// Mitsubishi GX Works2 project: auotomatation project   PLC: FX3G

// global labels: Global1
VAR_GLOBAL
  start_day AT X007 : BOOL;
  stock_oats AT D1100 : REAL;
  oats_input AT D1105 : REAL;
  stock_protein AT D2100 : REAL;
  protein_input AT D2105 : REAL;
  stock_honey AT D3100 : REAL;
  honey_input AT D3105 : REAL;
END_VAR
VAR_GLOBAL CONSTANT
  oats_min_need : REAL := 400;
  protein_min_need : REAL := 320;
  honey_min_need : REAL := 160;
END_VAR
VAR_GLOBAL
  enough_stock AT M1 : BOOL;
  valid_input AT M5 : BOOL;
  working AT Y000 : BOOL;
  emergency AT X005 : BOOL;
  Sample AT X003 : BOOL;
  Bar_Type AT D1160 : REAL;
END_VAR
VAR_GLOBAL CONSTANT
  Protein_Max : REAL := 10.0;
  Protein_Min : REAL := 5.0;
  Basic_Max : REAL := 5.0;
  Basic_Min : REAL;
END_VAR
VAR_GLOBAL
  Protein_Is_More_Beautiful AT M3 : BOOL;
  Basic_Is_Beautiful AT M4 : BOOL;
  MixingTime AT TC1 : BOOL;
END_VAR
VAR_GLOBAL CONSTANT
  MixingDuration : INT := 50;
END_VAR
VAR_GLOBAL
  EndMixing AT TS1 : BOOL;
  KeepOnMixingBaby AT Y003 : BOOL;
END_VAR
VAR_GLOBAL CONSTANT
  OATFOR8 : REAL := 400;
  OATFOR8PROTEIN : REAL := 240.0;
  ProteinFor8BASIC : REAL := 160.0;
  ProteinFor8 : REAL := 320.0;
  HoneyFor8Basic : REAL := 120.0;
  HoneyFor8 : REAL := 160.0;
  MixingFor8Basic : REAL := 680.0;
  MixingFor8Protein : REAL := 720.0;
END_VAR
VAR_GLOBAL
  MixingContainer AT D1150 : REAL;
  StartBake AT X002 : BOOL;
  BakeContainer AT D1170 : REAL;
  TimeForBakingB AT TC2 : BOOL;
  TimeForBakingP AT TC3 : BOOL;
  FinishBakingBasic AT TS2 : BOOL;
  FinishBakingProtein AT TS3 : BOOL;
  BlinkAssist AT M11 : BOOL;
  FirstLight AT TS4 : BOOL;
  Sirugin1 AT TC4 : BOOL;
  FirstBake AT Y001 : BOOL;
END_VAR
VAR_GLOBAL CONSTANT
  Sirugin : INT := 6;
END_VAR
VAR_GLOBAL
  Sirugin2 AT TC5 : BOOL;
  SecondLight AT TS5 : BOOL;
  SecondBake AT Y002 : BOOL;
  StartPacking AT X006 : BOOL;
  PackOneBar AT X000 : BOOL;
  CountFirstBar AT CC0 : BOOL;
END_VAR
VAR_GLOBAL CONSTANT
  CountedFirstBar : INT := 1;
END_VAR
VAR_GLOBAL
  Count8Bars AT CC1 : BOOL;
END_VAR
VAR_GLOBAL CONSTANT
  Counted8Bars : INT := 8;
END_VAR
VAR_GLOBAL
  BeginCount AT CS0 : BOOL;
  FinishCount AT CS1 : BOOL;
  AsLongAsPacking AT Y004 : BOOL;
  UpdateRegistryPacking AT Y004 : BOOL;
  SumOfPackges AT D1180 : REAL;
END_VAR
VAR_GLOBAL CONSTANT
  AddPack : REAL := 1.0;
END_VAR
VAR_GLOBAL
  FinishCount8Bars AT CS8 : BOOL;
  storage AT D5100 : REAL;
END_VAR
VAR_GLOBAL CONSTANT
  BarsBox : REAL := 1.0;
  convert_to_analog : REAL := 10.0;
END_VAR
VAR_GLOBAL
  enough_stock_another_iteration AT M2 : BOOL;
  enough_stock_to_start_day AT M1 : BOOL;
END_VAR
VAR_GLOBAL CONSTANT
  BakingDurationBasic : INT := 40;
  BakingDurationProtein : INT := 50;
END_VAR
VAR_GLOBAL
  FinishInterition AT M10 : BOOL;
  BlinkHelper AT M11 : BOOL;
END_VAR
VAR_GLOBAL CONSTANT
  OATFORPACK : REAL := 400.0;
END_VAR
VAR_GLOBAL
  CountTheFirstBar AT CC0 : BOOL;
END_VAR
VAR_GLOBAL CONSTANT
  CounterTheFirstBar : INT := 1;
END_VAR
VAR_GLOBAL
  CountThePack AT CC1 : BOOL;
END_VAR
VAR_GLOBAL CONSTANT
  CountedThePack : INT := 8;
END_VAR
VAR_GLOBAL
  CountBegan AT CS0 : BOOL;
  CountFinish AT CS1 : BOOL;
  analog_output AT D8282 : INT;
END_VAR
VAR_GLOBAL CONSTANT
  ten : REAL := 10.0;
END_VAR
VAR_GLOBAL
  AOutput AT D8282 : INT;
  SumOfPackgesWord AT D1190 : INT;
  Analog_Input1 AT D8280 : INT;
END_VAR
VAR_GLOBAL CONSTANT
  MitsubishiMagic : REAL := 400.0;
  MitsubishiMagic2 : REAL := 40.0;
END_VAR
VAR_GLOBAL
  SumOfPackgesOutPut AT D1190 : REAL;
END_VAR

// task Task_01 (event TRUE, interval 0, priority 31): POU_01

PROGRAM POU_01
(* structured ladder/FBD written out as ST: instructions are called as NAME(EN, inputs, outputs); _pN, _eN, _tN stand for wires *)
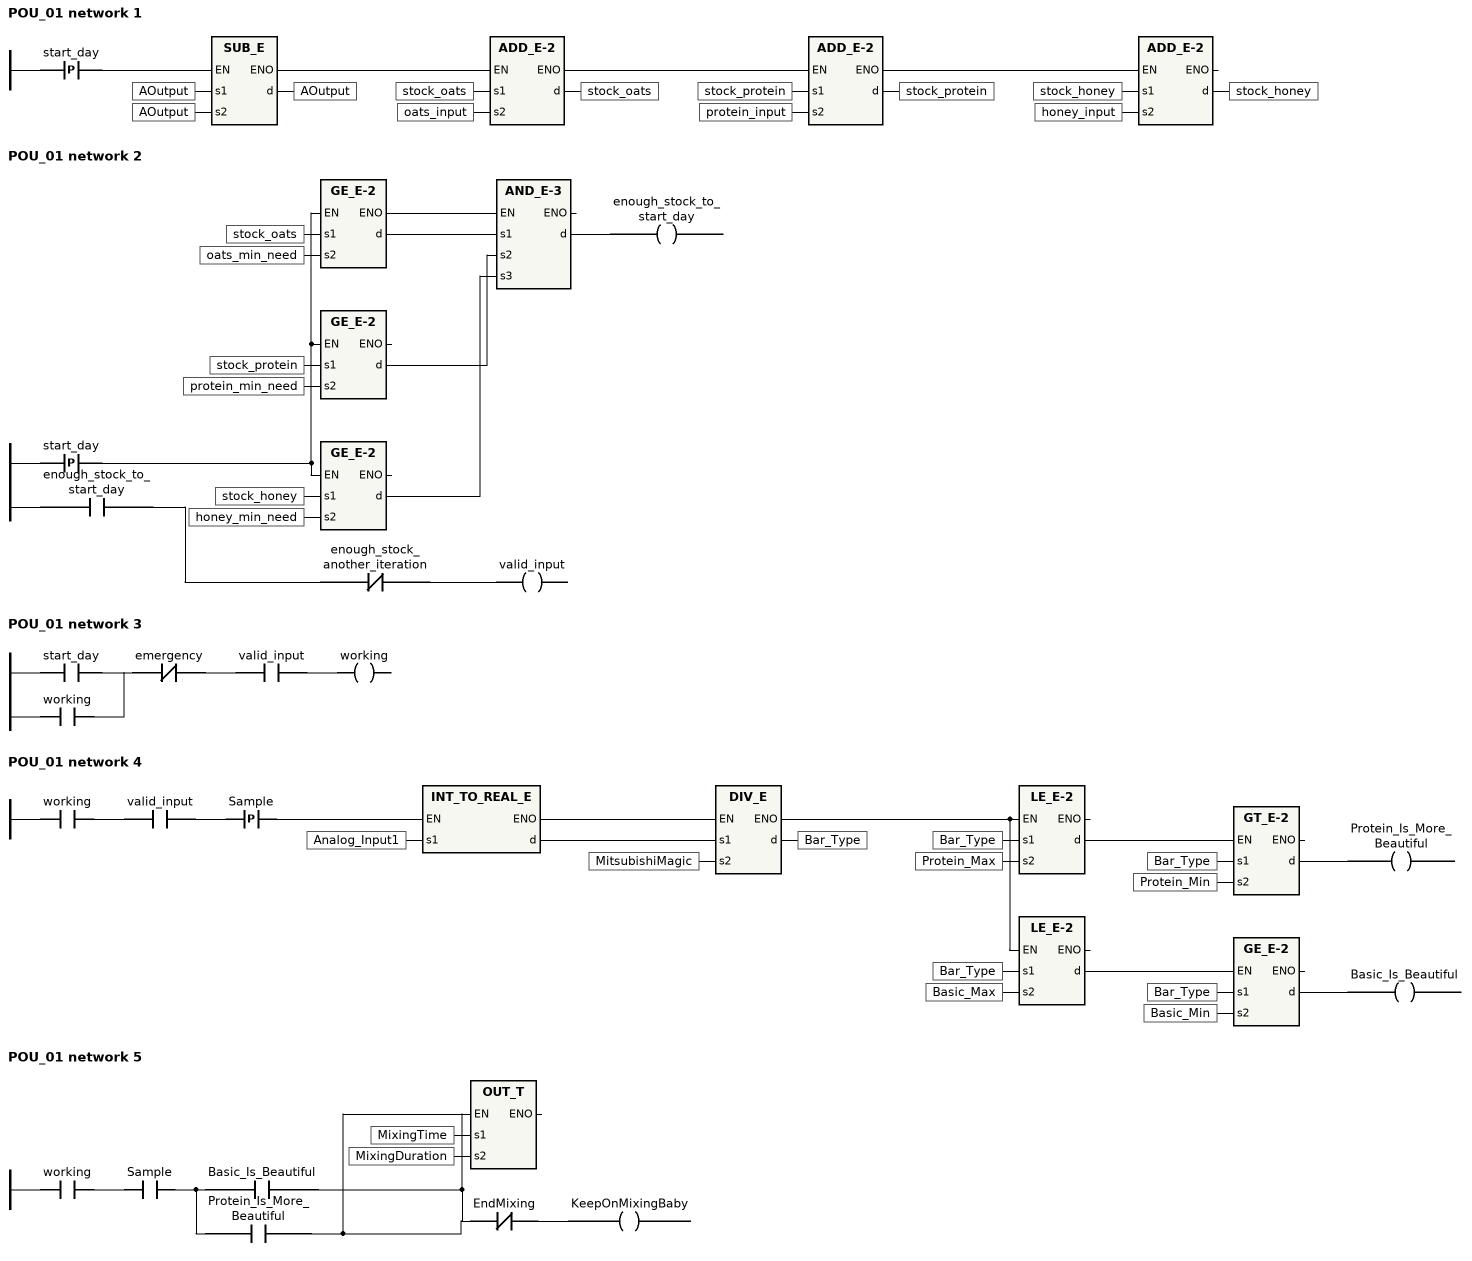
(* network 1 *)
_e1 := SUB_E(LDP(TRUE, start_day), AOutput, AOutput, AOutput);
_e2 := ADD_E(_e1, stock_oats, oats_input, stock_oats);
_e3 := ADD_E(_e2, stock_protein, protein_input, stock_protein);
ADD_E(_e3, stock_honey, honey_input, stock_honey);
(* network 2 *)
_p1 := LDP(TRUE, start_day);
_e3 := GE_E(_p1, stock_oats, oats_min_need, _t2);
GE_E(_p1, stock_protein, protein_min_need, _t4);
GE_E(_p1, stock_honey, honey_min_need, _t5);
AND_E(_e3, _t2, _t4, _t5, _t6);
enough_stock_to_start_day := _t6;
valid_input := enough_stock_to_start_day AND NOT enough_stock_another_iteration;
(* network 3 *)
working := ((start_day OR working) AND NOT emergency) AND valid_input;
(* network 4 *)
_e2 := INT_TO_REAL_E(working AND valid_input AND LDP(TRUE, Sample), Analog_Input1, _t1);
_e3 := DIV_E(_e2, _t1, MitsubishiMagic, Bar_Type);
LE_E(_e3, Bar_Type, Protein_Max, _t4);
GT_E(_t4, Bar_Type, Protein_Min, _t5);
Protein_Is_More_Beautiful := _t5;
LE_E(_e3, Bar_Type, Basic_Max, _t6);
GE_E(_t6, Bar_Type, Basic_Min, _t7);
Basic_Is_Beautiful := _t7;
(* network 5 *)
_p1 := working AND Sample;
_p2 := (_p1 AND Basic_Is_Beautiful) OR (_p1 AND Protein_Is_More_Beautiful);
OUT_T(_p2, MixingTime, MixingDuration);
KeepOnMixingBaby := _p2 AND NOT EndMixing;
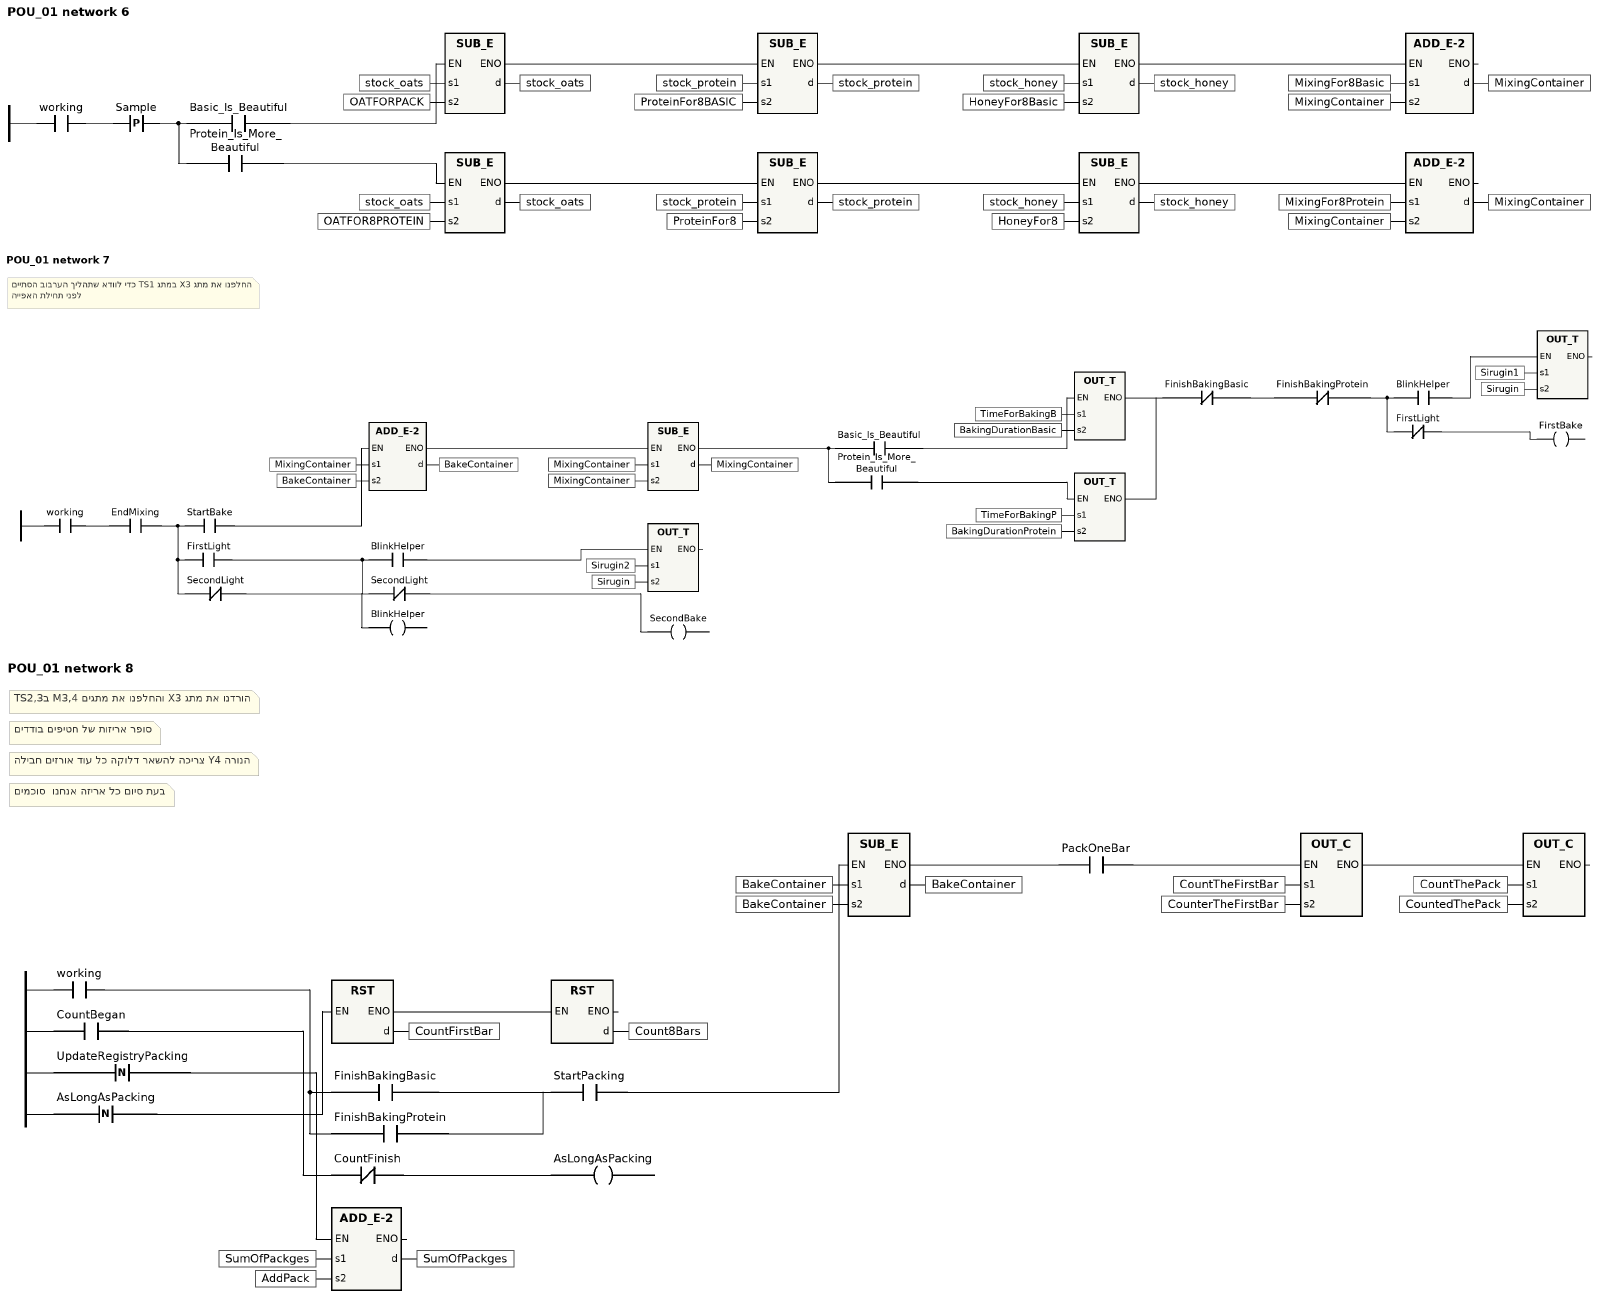
(* network 6 *)
_p1 := working AND LDP(TRUE, Sample);
_e2 := SUB_E(_p1 AND Basic_Is_Beautiful, stock_oats, OATFORPACK, stock_oats);
_e3 := SUB_E(_e2, stock_protein, ProteinFor8BASIC, stock_protein);
_e4 := SUB_E(_e3, stock_honey, HoneyFor8Basic, stock_honey);
ADD_E(_e4, MixingFor8Basic, MixingContainer, MixingContainer);
_e5 := SUB_E(_p1 AND Protein_Is_More_Beautiful, stock_oats, OATFOR8PROTEIN, stock_oats);
_e6 := SUB_E(_e5, stock_protein, ProteinFor8, stock_protein);
_e7 := SUB_E(_e6, stock_honey, HoneyFor8, stock_honey);
ADD_E(_e7, MixingFor8Protein, MixingContainer, MixingContainer);
(* network 7 *)
(* החלפנו את מתג X3 במתג TS1 כדי לוודא שתהליך הערבוב הסתיים לפני תחילת האפייה *)
_p1 := working AND EndMixing;
_e2 := ADD_E(_p1 AND StartBake, MixingContainer, BakeContainer, BakeContainer);
_e3 := SUB_E(_e2, MixingContainer, MixingContainer, MixingContainer);
_e4 := OUT_T(_e3 AND Basic_Is_Beautiful, TimeForBakingB, BakingDurationBasic);
_e5 := OUT_T(_e3 AND Protein_Is_More_Beautiful, TimeForBakingP, BakingDurationProtein);
_p6 := ((_e4 OR _e5) AND NOT FinishBakingBasic) AND NOT FinishBakingProtein;
OUT_T(_p6 AND BlinkHelper, Sirugin1, Sirugin);
FirstBake := _p6 AND NOT FirstLight;
_p7 := _p1 AND FirstLight;
OUT_T(_p7 AND BlinkHelper, Sirugin2, Sirugin);
SecondBake := _p7 AND NOT SecondLight;
BlinkHelper := _p1 AND NOT SecondLight;
(* network 8 *)
(* הורדנו את מתג X3 והחלפנו את מתגים M3,4 בTS2,3 *)
(* סופר אריזות של חטיפים בודדים *)
(* הנורה Y4 צריכה להשאר דלוקה כל עוד אורזים חבילה *)
(* בעת סיום כל אריזה אנחנו  סוכמים *)
_e1 := SUB_E(((working AND FinishBakingBasic) OR (working AND FinishBakingProtein)) AND StartPacking, BakeContainer, BakeContainer, BakeContainer);
_e2 := OUT_C(_e1 AND PackOneBar, CountTheFirstBar, CounterTheFirstBar);
OUT_C(_e2, CountThePack, CountedThePack);
AsLongAsPacking := CountBegan AND NOT CountFinish;
ADD_E(LDF(TRUE, UpdateRegistryPacking), SumOfPackges, AddPack, SumOfPackges);
_e3 := RST(LDF(TRUE, AsLongAsPacking), CountFirstBar);
RST(_e3, Count8Bars);
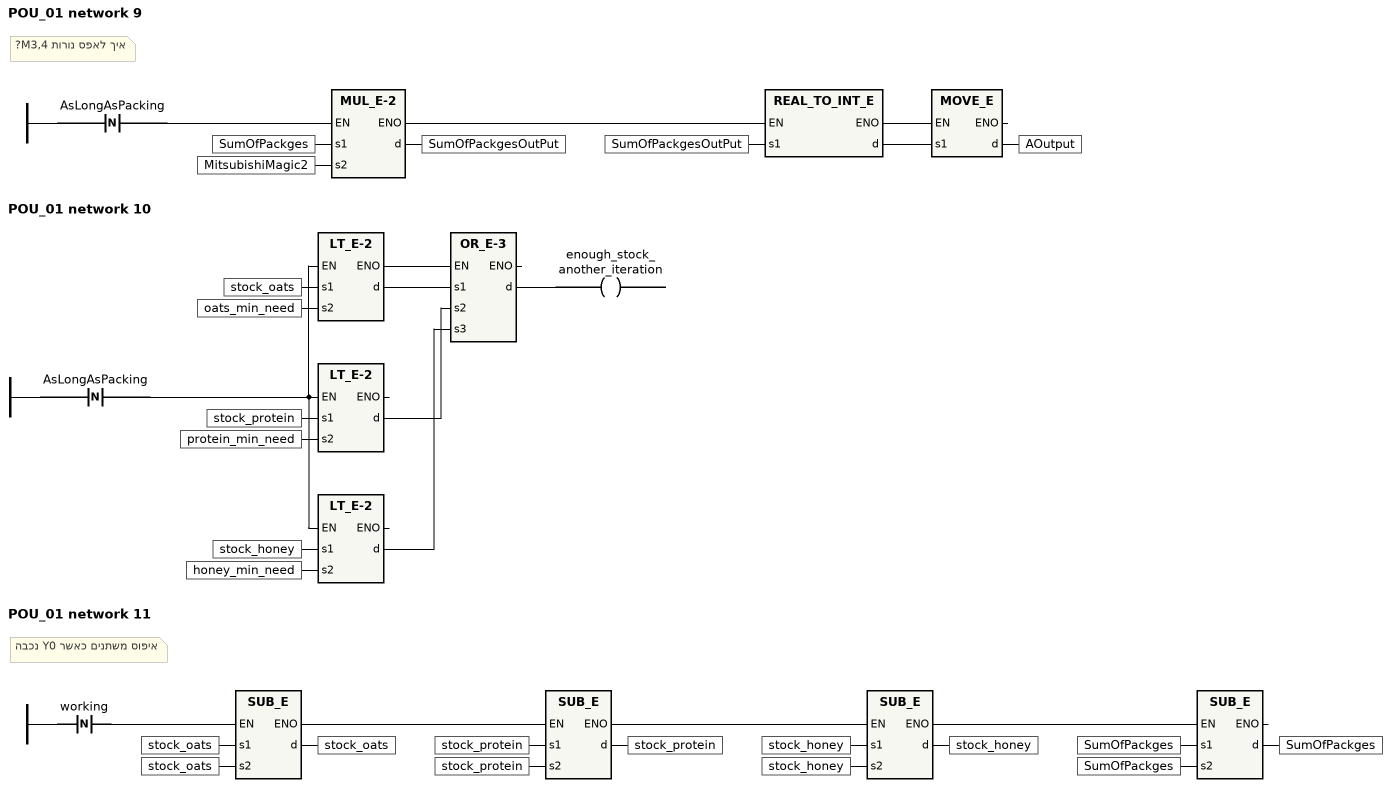
(* network 9 *)
(* איך לאפס נורות M3,4? *)
_e1 := MUL_E(LDF(TRUE, AsLongAsPacking), SumOfPackges, MitsubishiMagic2, SumOfPackgesOutPut);
_e3 := REAL_TO_INT_E(_e1, SumOfPackgesOutPut, _t2);
MOVE_E(_e3, _t2, AOutput);
(* network 10 *)
_p1 := LDF(TRUE, AsLongAsPacking);
_e3 := LT_E(_p1, stock_oats, oats_min_need, _t2);
LT_E(_p1, stock_protein, protein_min_need, _t4);
LT_E(_p1, stock_honey, honey_min_need, _t5);
OR_E(_e3, _t2, _t4, _t5, _t6);
enough_stock_another_iteration := _t6;
(* network 11 *)
(* איפוס משתנים כאשר Y0 נכבה *)
_e1 := SUB_E(LDF(TRUE, working), stock_oats, stock_oats, stock_oats);
_e2 := SUB_E(_e1, stock_protein, stock_protein, stock_protein);
_e3 := SUB_E(_e2, stock_honey, stock_honey, stock_honey);
SUB_E(_e3, SumOfPackges, SumOfPackges, SumOfPackges);
END_PROGRAM
